Universal Robots PolyScope program: rtde_control_loop.urp

Program rtde_control_loop (createdIn=3.2.19275.0 lastSavedIn=3.6.1.30595 robotSerialNumber=20235300917 directory=/home/ur/ursim-current/programs installation=default)
BeforeStart
  setp := p[0,0,0,0,0,0]
  Script: rtde_set_watchdog("input_int_register_0", 1, "PAUSE")
  Script: write_output_integer_register(0, 1)
Robot Program (runOnlyOnce=false motionType=MoveJ speed=1 acceleration=1.2 useActiveTCP=false)
  If read_input_integer_register(0)≟1 and setp≠p[0, 0, 0, 0, 0, 0]
    'Valid pose received from client'
    MoveJ speed 4.58 deg/s, acceleration 68.75 deg/s^2 (useActiveTCP=false) feature=Base
      Waypoint Waypoint (Variable): variable=setp
    'Confirm that move was executed'
    Script: write_output_integer_register(0, 0)
    'Wait until script acknowledges confirmation'
    Loop While (checkContinuously=false) expression=read_input_integer_register(0)≟1
      Script: sync()
    'Request next pose'
    Script: write_output_integer_register(0, 1)
  Script: sync()
Thread Thread_1 (runOnlyOnce=false trackProgramExecution=false)
  Loop Forever
    tmp := p[0,0,0,0,0,0]
    Script: tmp[0] = read_input_float_register(0)
    Script: tmp[1] = read_input_float_register(1)
    Script: tmp[2] = read_input_float_register(2)
    Script: tmp[3] = read_input_float_register(3)
    Script: tmp[4] = read_input_float_register(4)
    Script: tmp[5] = read_input_float_register(5)
    setp := tmp
    Script: sync()
